(* IEC 61131-3 sources: Slitting-Machine-Automation-Edge-Controller/firmware/build/ESP32-DOIT DEVKIT V1/src, 1 file *)

(* ---- program.st ---- *)
PROGRAM main
  VAR
    State : INT := 1;
    AutoStep : INT := 0;
    ton_Reset : TON;
    ton_Safeties : TON;
    ton_Start : TON;
    ton_Jam : TON;
    ton_EStop : TON;
    ton_Manual : TON;
    ton_PB1 : TON;
    ton_PB2 : TON;
    b_Reset : BOOL;
    b_SafetiesOK : BOOL;
    b_StartCycle : BOOL;
    b_JamDetected : BOOL;
    b_EStopPressed : BOOL;
    b_ManualMode : BOOL;
    b_PB1 : BOOL;
    b_PB2 : BOOL;
    ton_StepTimer : TON;
  END_VAR
  VAR
    i_SystemReset AT %IX0.0 : BOOL;
    i_SafetiesOK AT %IX0.1 : BOOL;
    i_StartCycle AT %IX0.2 : BOOL;
    i_JamDetected AT %IX0.3 : BOOL;
    i_EStopPressed AT %IX0.4 : BOOL;
    i_ManualMode AT %IX0.5 : BOOL;
    i_TwoHandPB1 AT %IX0.6 : BOOL;
    i_TwoHandPB2 AT %IX0.7 : BOOL;
    q_Pneumatics AT %QX0.0 : BOOL;
    q_Conveyor AT %QX0.1 : BOOL;
    q_Slitting AT %QX0.2 : BOOL;
    q_Offload AT %QX0.3 : BOOL;
    q_FaultLight AT %QX0.4 : BOOL;
  END_VAR

  // -----------------------------------------------------------------------------
  // 1. INPUT DEBOUNCING (50ms TON Timers for mechanical switch bounce)
  // -----------------------------------------------------------------------------
  ton_Reset(IN := i_SystemReset, PT := T#50MS, Q => b_Reset);
  ton_Safeties(IN := i_SafetiesOK, PT := T#50MS, Q => b_SafetiesOK);
  ton_Start(IN := i_StartCycle, PT := T#50MS, Q => b_StartCycle);
  ton_Jam(IN := i_JamDetected, PT := T#50MS, Q => b_JamDetected);
  ton_EStop(IN := i_EStopPressed, PT := T#50MS, Q => b_EStopPressed);
  ton_Manual(IN := i_ManualMode, PT := T#50MS, Q => b_ManualMode);
  ton_PB1(IN := i_TwoHandPB1, PT := T#50MS, Q => b_PB1);
  ton_PB2(IN := i_TwoHandPB2, PT := T#50MS, Q => b_PB2);

  // -----------------------------------------------------------------------------
  // 2. GLOBAL FAULT OVERRIDES
  // -----------------------------------------------------------------------------
  IF b_EStopPressed THEN
      State := 5; // Direct trip to E-STOP / FAULT
  ELSIF b_JamDetected AND (State = 3) THEN
      State := 4; // Jam Recovery triggered during AUTO RUN
  END_IF;

  // -----------------------------------------------------------------------------
  // 3. MAIN STATE MACHINE
  // -----------------------------------------------------------------------------
  CASE State OF

      1: // STOPPED STATE
          AutoStep := 0;
          IF b_Reset AND b_SafetiesOK THEN
              State := 2; // Transition to READY
          END_IF;

      2: // READY STATE
          IF b_StartCycle THEN
              State := 3; // Transition to AUTO RUN
              AutoStep := 1; // Start Step A
          ELSIF b_ManualMode THEN
              State := 6; // Transition to MANUAL / JOG
          END_IF;

      3: // AUTO RUN STATE (Sequential Steps A -> B -> C -> D with 5s Delays)
          CASE AutoStep OF
              1: // Step A: AGV Delivery & Robot Arm Load
                  ton_StepTimer(IN := TRUE, PT := T#5S);
                  IF ton_StepTimer.Q THEN
                      ton_StepTimer(IN := FALSE, PT := T#5S); // Reset Timer
                      AutoStep := 2; // Move to Step B
                  END_IF;

              2: // Step B: Conveyor Feed & Alignment
                  ton_StepTimer(IN := TRUE, PT := T#5S);
                  IF ton_StepTimer.Q THEN
                      ton_StepTimer(IN := FALSE, PT := T#5S); // Reset Timer
                      AutoStep := 3; // Move to Step C
                  END_IF;

              3: // Step C: Pneumatic Down-Clamp & Arbor Slitting
                  ton_StepTimer(IN := TRUE, PT := T#5S);
                  IF ton_StepTimer.Q THEN
                      ton_StepTimer(IN := FALSE, PT := T#5S); // Reset Timer
                      AutoStep := 4; // Move to Step D
                  END_IF;

              4: // Step D: Exit Sensing & Stacking Offload
                  ton_StepTimer(IN := TRUE, PT := T#5S);
                  IF ton_StepTimer.Q THEN
                      ton_StepTimer(IN := FALSE, PT := T#5S); // Reset Timer
                      State := 2; // Sequence Complete -> Return to READY
                  END_IF;
          END_CASE;

      4: // JAM RECOVERY STATE
          AutoStep := 0;
          ton_StepTimer(IN := FALSE, PT := T#5S);
          // Clearing jam transitions to STOPPED or MANUAL
          IF b_Reset THEN
              State := 1;
          ELSIF b_ManualMode THEN
              State := 6;
          END_IF;

      5: // E-STOP / FAULT STATE
          AutoStep := 0;
          ton_StepTimer(IN := FALSE, PT := T#5S);
          IF NOT b_EStopPressed AND b_ManualMode THEN
              State := 6; // Transition to MANUAL / JOG
          ELSIF NOT b_EStopPressed AND b_Reset THEN
              State := 1; // Return to STOPPED
          END_IF;

      6: // MANUAL / JOG STATE
          AutoStep := 0;
         // Transition out of Manual Mode using Reset or turning off Manual Mode
          IF b_Reset OR NOT b_ManualMode THEN
              State := 1; // Return to STOPPED
          END_IF;

  END_CASE;

  // Ensure timer resets if leaving state 3 prematurely
  IF State <> 3 THEN
      ton_StepTimer(IN := FALSE, PT := T#5S);
  END_IF;

  // -----------------------------------------------------------------------------
  // 4. OUTPUT MAPPING CONTROL
  // -----------------------------------------------------------------------------
  // Default outputs to FALSE
  q_Offload    := FALSE;
  q_Conveyor   := FALSE;
  q_Pneumatics := FALSE;
  q_Slitting   := FALSE;
  q_FaultLight := FALSE;

  CASE State OF
      3: // Outputs active sequentially based on AutoStep
          q_Offload    := (AutoStep = 1);
          q_Conveyor   := (AutoStep = 2);
          q_Pneumatics := (AutoStep = 3);
          q_Slitting   := (AutoStep = 4);

      4: // Jam Recovery: Release pneumatics
          q_Pneumatics := FALSE;
          q_FaultLight := TRUE; // Flash/Turn on fault indicator

      5: // E-Stop: Lock out system outputs, activate Fault Light
          q_FaultLight := TRUE;

      6: // Manual Control: Both PB1 and PB2 must be concurrently held
          IF b_PB1 AND b_PB2 THEN
              q_Slitting := TRUE; // Drives Arbor Slitting Machine
          END_IF;
  END_CASE;
END_PROGRAM

CONFIGURATION Config0

  RESOURCE Res0 ON PLC
    TASK task0(INTERVAL := T#20ms,PRIORITY := 1);
    PROGRAM instance0 WITH task0 : main;
  END_RESOURCE
END_CONFIGURATION
